FUNCTION_BLOCK E_CTUD
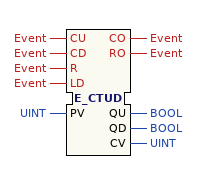
  EVENT_INPUT
    CU; (* Count Up *)
    CD; (* Count Down *)
    R; (* Reset *)
    LD; (* Load *)
  END_EVENT
  EVENT_OUTPUT
    CO; (* Carry Out *)
    RO; (* Reset Out *)
  END_EVENT
  VAR_INPUT
    PV : UINT; (* Preset Value *)
  END_VAR
  VAR_OUTPUT
    QU : BOOL; (* Up limit reached *)
    QD : BOOL; (* Down limit reached *)
    CV : UINT; (* Current Value *)
  END_VAR
END_FUNCTION_BLOCK
